(* IEC 61131-3 sources: plc_generation_empirical_study/datasets/task_bank_c06_bounded_runtime_v0_3/tasks/C06_U01_lean_composite/negative_control, 1 file *)

(* ---- NC1.st ---- *)
FUNCTION_BLOCK C06_U01_lean_composite
VAR_INPUT
    A_GoodPart : BOOL;
    A_RejectPart : BOOL;
    A_Reset : BOOL;
    A_BatchTarget : INT;
    A_RejectLimit : INT;
    B_Info : BOOL;
    B_Warning : BOOL;
    B_Trip : BOOL;
    B_Emergency : BOOL;
    B_Suppress : BOOL;
    SubsystemBEnable : BOOL;
    CrossReset : BOOL;
END_VAR
VAR_OUTPUT
    A_GoodCount : INT;
    A_RejectCount : INT;
    A_BatchDone : BOOL;
    A_QualityFault : BOOL;
    B_Active : BOOL;
    B_Level : INT;
    CrossReady : BOOL;
    CrossBlocked : BOOL;
END_VAR
VAR
    A_PrevGood : BOOL := FALSE;
    A_PrevReject : BOOL := FALSE;
END_VAR

IF A_Reset THEN
    A_GoodCount := 0;
    A_RejectCount := 0;
    A_QualityFault := FALSE;
ELSE
    IF A_RejectPart AND (NOT A_PrevReject) THEN
        A_RejectCount := A_RejectCount + 1;
    ELSIF A_GoodPart AND (NOT A_PrevGood) THEN
        A_GoodCount := A_GoodCount + 1;
    END_IF;
    IF A_RejectCount >= A_RejectLimit THEN
        A_QualityFault := TRUE;
    END_IF;
END_IF;
A_BatchDone := (A_GoodCount + A_RejectCount) >= A_BatchTarget;
A_PrevGood := A_GoodPart;
A_PrevReject := A_RejectPart;

IF CrossReset THEN
    CrossReady := FALSE;
ELSIF A_BatchDone THEN
    CrossReady := TRUE;
END_IF;
CrossBlocked := FALSE;

IF SubsystemBEnable AND CrossReady THEN
    IF B_Emergency THEN
        B_Level := 4;
        B_Active := TRUE;
    ELSIF B_Suppress THEN
        B_Level := 0;
        B_Active := FALSE;
    ELSIF B_Trip THEN
        B_Level := 3;
        B_Active := TRUE;
    ELSIF B_Warning THEN
        B_Level := 2;
        B_Active := TRUE;
    ELSIF B_Info THEN
        B_Level := 1;
        B_Active := TRUE;
    ELSE
        B_Level := 0;
        B_Active := FALSE;
    END_IF;
ELSE
    B_Active := FALSE;
    B_Level := 0;
END_IF;

END_FUNCTION_BLOCK
